# EPICS alarm handler configuration: mps_database/bareTest/alarms/areas/mpln_bpn22_mp01.alhConfig
GROUP NULL MPLN:BPN22:MP01:1
$ALIAS MPS Link Node 86
$GUIDANCE
LTUH MPS
   Group Name: MPLN:BPN22:MP01:1
   Summary PV:  MPLN:BPN22:MP01:1:STATSUMY
$END
CHANNEL  MPLN:BPN22:MP01:1    MPLN:BPN22:MP01:1:MPS_EN_RBV		-----
CHANNEL  MPLN:BPN22:MP01:1    MPLN:BPN22:MP01:1:LC1_MODE_RBV		-----
